// TIA Portal V20 export
TYPE "type_emRelations_em11_cmStatus"
// stored: Access Published, Namespace Unit1
   STRUCT
      WeightCheckJRDetect : "LBC_typeDigitalSignalControlNode";
      WeightCheckControl : "LER_WeightCheckControlNode";
   END_STRUCT;
END_TYPE
